FUNCTION_BLOCK StartingAborted (* Basic Function Block Type *)
  (* Standard: 61499-2 *)
  (* Version 0.0, 7/17/2026, Schneider Electric, Template *)
  PACKAGE SE.Nereda;
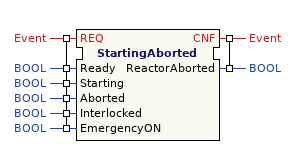
  EVENT_INPUT
    REQ WITH Starting, Aborted, Ready, Interlocked, EmergencyON; (* Normal Execution Request *)
  END_EVENT
  EVENT_OUTPUT
    CNF WITH ReactorAborted; (* Execution Confirmation *)
  END_EVENT
  VAR_INPUT
    Ready : BOOL;
    Starting : BOOL;
    Aborted : BOOL;
    Interlocked : BOOL;
    EmergencyON : BOOL;
  END_VAR
  VAR_OUTPUT
    ReactorAborted : BOOL;
  END_VAR
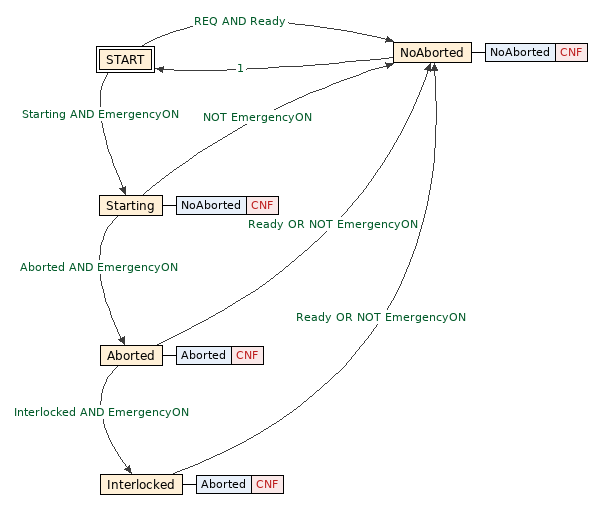
  EC_STATES
    START; (* Initial State *)
    Starting : NoAborted -> CNF; (* Normal execution *)
    Aborted : Aborted -> CNF;
    NoAborted : NoAborted -> CNF;
    Interlocked : Aborted -> CNF;
  END_STATES
  EC_TRANSITIONS
    START TO Starting := Starting AND EmergencyON;
    Starting TO Aborted := Aborted AND EmergencyON;
    Interlocked TO NoAborted := Ready OR NOT EmergencyON;
    START TO NoAborted := REQ AND Ready;
    NoAborted TO START := 1;
    Aborted TO Interlocked := Interlocked AND EmergencyON;
    Aborted TO NoAborted := Ready OR NOT EmergencyON;
    Starting TO NoAborted := NOT EmergencyON;
  END_TRANSITIONS
  ALGORITHM Aborted IN ST:
;
ReactorAborted := TRUE;
  END_ALGORITHM
  ALGORITHM NoAborted IN ST:
;
ReactorAborted := FALSE;
  END_ALGORITHM
END_FUNCTION_BLOCK
